# EPICS alarm handler configuration: alh_files/mgnt_li24.alhConfig
GROUP NULL MGNT:LI24:1
   $COMMAND edm -x -eolc -noedit mgnt_li24_main.edl

$ALIAS LI24
$GUIDANCE
li24 Magnets
   Group Name: MGNT:LI24:1
   Summary PV:  MGNT:LI24:1:STATSUMY
$END

   INCLUDE MGNT:LI24:1 ./mgnt_li24_bend.alhConfig
   INCLUDE MGNT:LI24:1 ./mgnt_li24_lgps.alhConfig
   INCLUDE MGNT:LI24:1 ./mgnt_li24_quad.alhConfig
   INCLUDE MGNT:LI24:1 ./mgnt_li24_xcor.alhConfig
   INCLUDE MGNT:LI24:1 ./mgnt_li24_ycor.alhConfig
